TYPE ST_CSV_Record :
STRUCT
	sName 		: T_MaxString 	:= '';
	nNumber		: UDINT 		:= 0;
	fPos		: LREAL 		:= 0.0;
	bOP			: BOOL 			:= FALSE;
	sDesc		: STRING(40)	:= '';
	data		: ARRAY[0..7] OF BYTE;
END_STRUCT
END_TYPE

(* stored: Version 1.1.0.1, ProductVersion 3.1.4022.12
   DUT ST_CSV_Record: Id {7b76f7a7-c581-46ac-8d54-525e2d3c3486} *)
